PROGRAM P_Demo_FB_HVACRedundancyCtrlEx
VAR
    fb : FB_HVACRedundancyCtrlEx;                            // 被演示 FB 实例
    eDataSecurityType_in : E_HVACDataSecurityType ;
    bSetDefault_in : BOOL := FALSE;
    iCountCtrl_in : INT := 0;
    bForceChange_in : BOOL := FALSE;
    tOverlap1Actuator_io : TIME := T#0S;
    uiMaxOnLevel_io : UINT := 0;
    tNoFeedbActuator_io : TIME := T#0S;
    arrFiFo_out : Array[1..8] of INT;
    eErrorCode_out : E_HVACErrorCodes;
    bErrorGeneral_out : BOOL;
    bInvalidParameter_out : BOOL;
END_VAR

// ============================================================================
// Tc2_HVAC.FB_HVACRedundancyCtrlEx 演示程序
// ============================================================================
// 场景：把本 FB 实例化到一个 PLC 程序里，每周期单次调用；按需要把 VAR_INPUT 与
//       VAR_IN_OUT 接到工程信号；VAR_OUTPUT 写入对应监视变量。
// 价值：使用本 FB 比手写状态机 / 控制算法节省大量代码；与 Tc2_HVAC 体系内其它 FB
//       直接对接，命名 / 持久化 / 模式仲裁等约定一致。具体语义见 FB_HVACRedundancyCtrlEx.md 主文档。
// 验证步骤：
//   1. 右键 PLC 项目下 POUs 文件夹 → Add → Existing Item → 选本 .TcPOU 文件
//   2. 引用 Tc2_HVAC（References → Add library）
//   3. 编译 → 登录 → 运行
//   4. 在线写各 *_in 输入信号触发 FB；在线 monitor *_out 引脚观察状态
// ============================================================================

fb(
    eDataSecurityType := eDataSecurityType_in,
    bSetDefault := bSetDefault_in,
    iCountCtrl := iCountCtrl_in,
    bForceChange := bForceChange_in,
    tOverlap1Actuator := tOverlap1Actuator_io,
    uiMaxOnLevel := uiMaxOnLevel_io,
    tNoFeedbActuator := tNoFeedbActuator_io,
    arrFiFo => arrFiFo_out,
    eErrorCode => eErrorCode_out,
    bErrorGeneral => bErrorGeneral_out,
    bInvalidParameter => bInvalidParameter_out
);

END_PROGRAM

(* stored: Version 1.1.0.1, ProductVersion 3.1.4024.5
   POU P_Demo_FB_HVACRedundancyCtrlEx: Id {5df1ca2f-f028-54ed-8b20-aedb93e16213}, SpecialFunc None *)
